// TwinCAT 3 PLC project Queque
// ProgramVersion: 3.1.0.9
// libraries:
//   CAA Memory, * (CAA Technical Workgroup)
//   VisuElem3DPath, 3.5.6.0 (System)
//   VisuElemMeter, 3.5.6.0 (System)
//   VisuElems, 3.5.6.10 (System)
//   VisuElemsDateTime, 3.5.6.0 (System)
//   VisuElemsSpecialControls, 3.5.6.0 (System)
//   VisuElemsWinControls, 3.5.6.0 (System)
//   VisuElemTextEditor, 3.5.6.0 (System)
//   visuinputs, 3.5.6.0 (system)
//   VisuNativeControl, 3.5.6.0 (System)
//   Tc2_MC2, * (Beckhoff Automation GmbH)
//   Tc2_Standard, * (Beckhoff Automation GmbH)
//   Tc2_System, * (Beckhoff Automation GmbH)
//   Tc2_TcpIp, * (Beckhoff Automation GmbH)
//   Tc2_Utilities, * (Beckhoff Automation GmbH)
//   Tc3_Interfaces, * (Beckhoff Automation GmbH)
//   Tc3_Module, * (Beckhoff Automation GmbH)
// project tree:
//   DUTs/enum/ ENUM_REC_FUNCTION_CODE.TcDUT
//   DUTs/struct/ ERROR_RECORD.TcDUT
//   / GlobalTextList.TcGTLO (not stored), PlcTask.TcTTO, Visualization Manager.TcVMO (not stored)
//   GVLs/ Error_Record_Data.TcGVL (not stored), MachineData.TcGVL (not stored)
//   POUs/AxisContrl/ Axis_Contrl.TcPOU
//   POUs/ CMD_Manage.TcPOU, Err_Record.TcPOU, IOInstances_Axis.TcPOU, IOInstances_Cylinder.TcPOU, MAIN.TcPOU (not stored), Param_Queue.TcGVL, P_TextModeWrite.TcPOU (not stored), Queue_REC_Contrl.TcPOU, Queue_SEND_Contrl.TcPOU
//   POUs/CMD_Manager_Ctrl/ CMD_Manager.TcPOU
//   POUs/CylinderContrl/ Cylinder_Contrl.TcPOU (not stored)
//   POUs/DUTs_Queue/ REC_CMD_DATA.TcDUT (not stored), REC_iCMD_DATA.TcDUT (not stored), SEND_CMD_DATA.TcDUT (not stored), SEND_iCMD_DATA.TcDUT
//   POUs/Queue_Ctrl/ Rec_Queue.TcPOU (not stored), Send_Queue.TcPOU (not stored)
//   POUs/TCP/ Client.TcPOU (not stored), Server.TcPOU
//   VISUs/ Axis_HMI_Struct.TcDUT, Axis_Page.TcVIS (not stored), CtrlMode_List.TcTLO, Cylinder.TcVIS, Cylinder_HMI_Structure.TcDUT (not stored), Err_record.TcVIS (not stored), Main.TcVIS

CONFIGURATION Queque
    RESOURCE PLC ON TwinCAT3
        TASK PlcTask(INTERVAL := T#10ms, PRIORITY := 20);
        PROGRAM MAIN WITH PlcTask : MAIN;
    END_RESOURCE
END_CONFIGURATION

// ---- DUTs/enum/ENUM_REC_FUNCTION_CODE.TcDUT
TYPE ENUM_REC_FUNCTION_CODE :
(
	(*__________Axis Control_________________*)
	MD  := 0,//Digital
	MA  := 1,//Analog
	G00 := 2,//move absolute
	G01 := 3,//move relative
	G02 := 4,//move velocity
	G03 := 5,//move Jog
	G04 := 6,//go home
	G05 := 7,//reset error
	G06 := 8,//stop
	
   (*________Cylinder Control_______________*)	
	C00 := 10,// Extend
	C01 := 11,// Retract
	C02 := 12 // Reset
)UDINT;
END_TYPE

// ---- DUTs/struct/ERROR_RECORD.TcDUT
TYPE ERROR_RECORD :
STRUCT
	Timer       : STRING;
	Axis        : UDINT;
	ErrorID     : UDINT;
	ErrorTXT    : STRING;
	ErrorCNT    : UDINT:=0;
END_STRUCT
END_TYPE

// ---- POUs/DUTs_Queue/SEND_iCMD_DATA.TcDUT
TYPE SEND_iCMD_DATA :
STRUCT
	DEVICE_ID       : UDINT;
	FUNCTIONCODE    : UDINT;
	DATA            : LREAL;
	Vel             : LREAL;
END_STRUCT
END_TYPE

// ---- VISUs/Axis_HMI_Struct.TcDUT
TYPE Axis_HMI_Struct :
STRUCT
	(*-------- input----------------*)
	mode                     : UDINT;
	bStop_Man                : BOOL;
	bHalt_Man                : BOOL;
	bReset_Man               : BOOL;
	bJog_F                   : BOOL;
	bJog_B                   : BOOL;
	bAbsGo_Man               : BOOL;
	bAddGo_Man               : BOOL;
	bVelGo_Man               : BOOL;
	bRelGo_Man               : BOOL;
	bModGo_Man               : BOOL;
	fSetAbsPos_Man           : LREAL;
	fSetRelPos_Man           : LREAL;
	fSetModPos_Man           : LREAL;
	fSetVel_Man              : LREAL;
	softLimitPOS_FW          : LREAL;
	softLimitPOS_BW          : LREAL;
	bForwordEnable           : BOOL;
	bBackwordEnable          : BOOL;
	bFW_LimitSwith           : BOOL;
	bBW_LimitSwith           : BOOL;
	bDog_PointSwith          : BOOL;

	(*---------output-------------*)
	bPowerEn                 : BOOL;
	bBusy                    : BOOL;
	bDone                    : BOOL;
	bAborted                 : BOOL;
	bError                   : BOOL;
	nErrorID                 : UDINT;
	cErrorTXT                : STRING;
	
	Axis_ref                 : Axis_ref;
END_STRUCT
END_TYPE

// ---- POUs/Param_Queue.TcGVL
VAR_GLOBAL CONSTANT
	MAX_QUEUE_SIZE : INT:= 10;

END_VAR

// ---- POUs/AxisContrl/Axis_Contrl.TcPOU
FUNCTION_BLOCK Axis_Contrl
VAR_IN_OUT
	HMI                      : Axis_HMI_Struct;
	Axis_CMD_Itf             : REC_CMD_DATA;
	Axis_ref                 : axis_ref;
END_VAR
VAR_INPUT
	mode                     : UDINT;
	bStop_Man                : BOOL;
	bStop_Auto               : BOOL;
	bHalt_Man                : BOOL;
	bReset_Man               : BOOL;
	bReset_Auto              : BOOL;
	bJog_F                   : BOOL;
	bJog_B                   : BOOL;
	bAbsGo_Man               : BOOL;
	bAbsGo_Auto              : BOOL;
	bVelGo_Man               : BOOL;
	bVelGo_Auto              : BOOL;
	bRelGo_Man               : BOOL;
	bRelGo_Auto              : BOOL;
	bModGo_Man               : BOOL;
	bModGo_Auto              : BOOL;
	bAddGo_Man               : BOOL;
	fSetAbsPos_Man           : LREAL;
	fSetAbsPos_Auto          : LREAL;
	fSetRelPos_Man           : LREAL;
	fSetRelPos_Auto          : LREAL;
	fSetModPos_Man           : LREAL;
	fSetModPos_Auto          : LREAL;
	fSetVel_Man              : LREAL;
	fSetVel_Auto             : LREAL;
	softLimitPOS_FW          : LREAL;
	softLimitPOS_BW          : LREAL;
	bForwordEnable           : BOOL:= TRUE;
	bBackwordEnable          : BOOL:= TRUE;
	bFW_LimitSwith           : BOOL:= TRUE;
	bBW_LimitSwith           : BOOL:= TRUE;
	bDog_PointSwith          : BOOL;
END_VAR
VAR_OUTPUT
	bPowerEn                 : BOOL;
	bBusy                    : BOOL;
	bDone                    : BOOL;
	bAborted                 : BOOL;
	bError                   : BOOL;
	nErrorID                 : UDINT;
	cErrorTXT                : STRING;
	nStatus                  : STRING;
END_VAR	
VAR

	mc_Stop                  : MC_Stop;
	mc_Reset                 : MC_Reset;
	mc_Power                 : MC_Power;
	mc_Jog                   : MC_Jog;
	mc_Home                  : MC_Home;
	mc_AbsMove               : MC_MoveAbsolute;
	mc_VelMove               : MC_MoveVelocity;
	mc_RelMove               : MC_MoveRelative;
	mc_ModMove               : MC_MoveModulo;
	mc_ReadAxisError         : MC_ReadAxisError;
	
	mc_AddMove               : MC_MoveAdditive;
	mc_Halt                  : MC_Halt;
	
	
	AbsMove_Rtrig            : R_Trig;
	VelMove_Rtrig            : R_Trig;
	RelMove_Rtrig            : R_Trig;
	ModMove_Rtrig            : R_Trig;

	
	AbsMove_state            : INT;
	VelMove_state            : INT;
	RelMove_state            : INT;
	ModMove_state            : INT;
	
	
	CMD_state                : UDINT;
END_VAR

Axis_AbsMove();
Axis_AddMove();
Axis_Home();
Axis_Jog();
Axis_ModMove();
Axis_Power();
Axis_RelMove();
Axis_Reset();
Axis_Stop();
Axis_VelMove();
HMI_Mapping();
Read_AxisError();
Axis_Halt();
Queue_Rec_Cmd();
//---------------------------------------
IF bError THEN
	nStatus:='ERROR';
ELSIF bDone AND (NOT bBusy) THEN
	nStatus:='DONE';
ELSIF Main.sReceiveData.Delete_Queue.FUNCTIONCODE = G05 THEN
	nStatus:= 'RESET DONE';
ELSE
	nStatus:= '';
END_IF

METHOD Axis_AbsMove
VAR_INPUT
END_VAR
mc_AbsMove( Axis:= Axis_ref );

IF ((bReset_Man OR bReset_Auto) AND (bError OR NOT mc_AbsMove.Busy)) 
	OR bStop_Auto OR bStop_Man  THEN
	mc_AbsMove.Execute:= FALSE;
	AbsMove_state:= 0;
END_IF

CASE mode OF
	1:
		mc_AbsMove.Position := fSetAbsPos_Man;
		mc_AbsMove.Velocity := ABS(fSetVel_Man);	
	2:
		mc_AbsMove.Position := fSetAbsPos_Auto;
		mc_AbsMove.Velocity := ABS(fSetVel_Auto);	
END_CASE

AbsMove_Rtrig(CLK:= ((mode = 1) AND bAbsGo_Man) OR ((mode = 2) AND bAbsGo_Auto) );

CASE AbsMove_state OF
	0:	
    	mc_AbsMove.Execute:= FALSE;
		IF AbsMove_Rtrig.Q THEN
			IF (NOT bForwordEnable) OR (NOT bBackwordEnable) 
				OR (mc_AbsMove.Position > softLimitPOS_FW) 
				OR (mc_AbsMove.Position < softLimitPOS_BW) 
				OR (NOT bFW_LimitSwith) OR (NOT bBW_LimitSwith)
				OR bError
				THEN
				bError:= TRUE;
				bBusy:= FALSE;
				bDone:= FALSE;
				bAborted:= FALSE;
				IF (NOT bForwordEnable) OR (NOT bBackwordEnable) THEN
					nErrorID:= 1;
					cErrorTXT:= 'Error: Axis not enable';
				ELSIF (mc_AbsMove.Position > softLimitPOS_FW) OR
					  (mc_AbsMove.Position < softLimitPOS_BW) THEN
					nErrorID:= 2;
					cErrorTXT:= 'Error: Axis Absolute Movement out of Limits';
				ELSIF (NOT bFW_LimitSwith) OR (NOT bBW_LimitSwith) THEN
					nErrorID:= 3;
					cErrorTXT:= 'Error: Axis reach limit swith';
				END_IF
			ELSE
				bBusy:= TRUE;
				bDone:= FALSE;
				bAborted:= FALSE;
				bError:= FALSE;
				nErrorID:= 0;
				cErrorTXT:= '';	
				AbsMove_state:= 1;
			END_IF
		END_IF
	1:
		mc_AbsMove.Execute:= TRUE;
		IF mc_AbsMove.Error THEN
			mc_AbsMove.Execute:= FALSE;
			bError:= TRUE;
			bAborted:= FALSE;
			bBusy:= FALSE;
			bDone:= FALSE;
			nErrorID:= DWORD_TO_UDINT (mc_AbsMove.ErrorID);
			cErrorTXT:= 'Error: Axis absolute movement error';
			AbsMove_state:= 0;
		ELSIF (NOT bFW_LimitSwith) OR (NOT bBW_LimitSwith) THEN
			mc_AbsMove.Execute:= FALSE;
			bError:= TRUE;
			bAborted:= FALSE;
			bBusy:= FALSE;
			bDone:= FALSE;
			nErrorID:= 3;
			cErrorTXT:= 'Error: Axis reach limit swith';
			AbsMove_state:= 0;
		ELSIF mc_AbsMove.Done THEN
			mc_AbsMove.Execute:= FALSE;
			bDone:= TRUE;
			bAborted:= FALSE;
			bBusy:= FALSE;
			AbsMove_state:= 0;
		ELSIF mc_AbsMove.CommandAborted THEN
			mc_AbsMove.Execute:= FALSE;
			bAborted:= TRUE;
			bDone:= FALSE;
			bBusy:= FALSE;
			AbsMove_state:= 0;
		END_IF
END_CASE
END_METHOD

METHOD Axis_AddMove
VAR_INPUT
END_VAR
mc_AddMove(
	Axis:=Axis_ref , 
	Execute:=bAddGo_Man , 
	Distance:=fSetRelPos_Man , 
	Velocity:= ABS(fSetVel_Man) , 
	Acceleration:= , 
	Deceleration:= , 
	Jerk:= , 
	BufferMode:= , 
	Options:= , 
	Done=> , 
	Busy=> , 
	Active=> , 
	CommandAborted=> , 
	Error=> , 
	ErrorID=> );
END_METHOD

METHOD Axis_Halt
VAR_INPUT
END_VAR
mc_Halt(
	Axis:= Axis_ref , 
	Execute:= bHalt_Man , 
	Deceleration:= , 
	Jerk:= , 
	BufferMode:= , 
	Options:= , 
	Done=> , 
	Busy=> , 
	Active=> , 
	CommandAborted=> , 
	Error=> , 
	ErrorID=> );
END_METHOD

METHOD Axis_Home
VAR_INPUT
END_VAR
mc_Home(
	Axis:= Axis_ref , 
	Position:= , 
	HomingMode:= MC_Direct , 
	bCalibrationCam:= bDog_PointSwith , 
	 );
	 
IF ((bReset_Man OR bReset_Auto) AND (bError OR NOT mc_Home.Busy)) 
	OR bStop_Auto OR bStop_Man  THEN
	mc_Home.Execute:= FALSE;
END_IF
END_METHOD

METHOD Axis_Jog
VAR_INPUT
END_VAR
mc_Jog(
	Axis:= Axis_ref , 
	JogForward:= bJog_F AND (mode = 1) AND bForwordEnable AND bFW_LimitSwith AND NOT bError , 
	JogBackwards:= bJog_B AND (mode = 1) AND bBackwordEnable AND bBW_LimitSwith AND NOT bError, 
	Mode:= MC_JOGMODE_CONTINOUS , 
	Position:= , 
	Velocity:= fSetVel_Man, 
	 );
END_METHOD

METHOD Axis_ModMove
VAR_INPUT
END_VAR
mc_ModMove( Axis:= Axis_ref , Direction:= MC_Shortest_Way );

IF ((bReset_Man OR bReset_Auto) AND (bError OR NOT mc_ModMove.Busy)) 
	OR bStop_Auto OR bStop_Man  THEN
	mc_ModMove.Execute:= FALSE;
	ModMove_state:= 0;
END_IF

CASE mode OF
	1:
		mc_ModMove.Velocity:= ABS(fSetVel_Man);
		mc_ModMove.Position:= fSetModPos_Man;
	2:
		mc_ModMove.Velocity:= ABS(fSetVel_Auto);
		mc_ModMove.Position:= fSetModPos_Auto;
END_CASE

ModMove_Rtrig(CLK:= ((mode = 1) AND bModGo_Man) OR ((mode = 2) AND bModGo_Auto) );

CASE ModMove_state OF
	0:
		mc_ModMove.Execute:= FALSE;
		IF ModMove_Rtrig.Q THEN
			IF (NOT bForwordEnable) OR (NOT bBackwordEnable) 
				OR (NOT bFW_LimitSwith) OR (NOT bBW_LimitSwith)
				OR bError
				THEN
				bError:= TRUE;
				bBusy:= FALSE;
				bDone:= FALSE;
				bAborted:= FALSE;
				IF (NOT bForwordEnable) OR (NOT bBackwordEnable) THEN
					nErrorID:= 1;
					cErrorTXT:= 'Error: Axis not enable';
				ELSIF (NOT bFW_LimitSwith) OR (NOT bBW_LimitSwith) THEN
					nErrorID:= 3;
					cErrorTXT:= 'Error: Axis reach limit swith';
				END_IF
			ELSE 
				bBusy:= TRUE;
				bDone:= FALSE;
				bAborted:= FALSE;
				bError:= FALSE;
				nErrorID:= 0;
				cErrorTXT:= '';	
				ModMove_state:= 1;
			END_IF
		END_IF
	1:
		mc_ModMove.Execute:= TRUE;
		IF mc_ModMove.Error THEN
			mc_ModMove.Execute:= FALSE;
			bError:= TRUE;
			bBusy:= FALSE;
			bDone:= FALSE;
			bAborted:= FALSE;
			nErrorID:= DWORD_TO_UDINT(mc_ModMove.ErrorID);
			cErrorTXT:= 'Error: Axis Modulo Movement error';
			ModMove_state:= 0;
		ELSIF (NOT bFW_LimitSwith) OR (NOT bBW_LimitSwith) THEN
			mc_AbsMove.Execute:= FALSE;
			bError:= TRUE;
			bAborted:= FALSE;
			bBusy:= FALSE;
			bDone:= FALSE;
			nErrorID:= 3;
			cErrorTXT:= 'Error: Axis reach limit swith';		
		ELSIF mc_ModMove.Done THEN
			mc_ModMove.Execute:= FALSE;
			bDone:= TRUE;
			bBusy:= FALSE;
			bAborted:= FALSE;
			ModMove_state:= 0;
		ELSIF mc_ModMove.CommandAborted THEN
			mc_ModMove.Execute:= FALSE;
			bAborted:= TRUE;
			bBusy:= FALSE;
			bDone:= FALSE;
			ModMove_state:= 0;
		END_IF
END_CASE
END_METHOD

METHOD Axis_Power
VAR_INPUT
END_VAR

mc_Power(
	Axis:= Axis_ref , 
	Enable:= TRUE , 
	Enable_Positive:= bFW_LimitSwith AND bForwordEnable , 
	Enable_Negative:= bBW_LimitSwith AND bBackwordEnable, 
	Override:=100.0 , 
	BufferMode:= , 
	Options:= , 
	Status=> bPowerEn , 
	Busy=> , 
	Active=> , 
	Error=> , 
	ErrorID=> );
END_METHOD

METHOD Axis_RelMove
VAR_INPUT
END_VAR
mc_RelMove(Axis:= Axis_ref);

IF ((bReset_Man OR bReset_Auto) AND (bError OR NOT mc_RelMove.Busy ))
	OR bStop_Man OR bStop_Auto THEN
	mc_RelMove.Execute:= FALSE;
	RelMove_state:= 0;
END_IF

CASE mode OF
	1:
		mc_RelMove.Velocity:= ABS(fSetVel_Man);
		mc_RelMove.Distance:= fSetRelPos_Man;
	2:
		mc_RelMove.Velocity:= ABS(fSetVel_Auto);
		mc_RelMove.Distance:= fSetRelPos_Auto;
END_CASE

RelMove_Rtrig(CLK:= ((mode = 1) AND bRelGo_Man) OR ((mode = 2) AND bRelGo_Auto) );

CASE RelMove_state OF
	0:
		mc_RelMove.Execute:= FALSE;
		IF RelMove_Rtrig.Q THEN
			IF (NOT bForwordEnable) OR (NOT bBackwordEnable) 
				OR ((mc_RelMove.Distance + Axis_ref.NcToPlc.ActPos) > softLimitPOS_FW) 
				OR ((mc_RelMove.Distance + Axis_ref.NcToPlc.ActPos) < softLimitPOS_BW)
				OR (NOT bFW_LimitSwith) OR (NOT bBW_LimitSwith)
				OR bError
				THEN
				bError:= TRUE;
				bAborted:= FALSE;
				bBusy:= FALSE;
				bDone:= FALSE;
				IF (NOT bForwordEnable) OR (NOT bBackwordEnable) THEN
					nErrorID:= 1;
					cErrorTXT:= 'Error: Axis not enable';
				ELSIF ((mc_RelMove.Distance + Axis_ref.NcToPlc.ActPos) > softLimitPOS_FW)
				    OR ((mc_RelMove.Distance + Axis_ref.NcToPlc.ActPos) < softLimitPOS_BW) THEN
					nErrorID:= 2;
					cErrorTXT:= 'Error: Axis Relative movement out of limits';
				ELSIF (NOT bFW_LimitSwith) OR (NOT bBW_LimitSwith) THEN
					nErrorID:= 3;
					cErrorTXT:= 'Error: Axis reach limit swith';
				END_IF
			ELSE
				bBusy:= TRUE;
				bDone:= FALSE;
				bAborted:= FALSE;
				bError:= FALSE;
				nErrorID:= 0;
				cErrorTXT:= '';	
				RelMove_state:= 1;
			END_IF
		END_IF
	1: 
		mc_RelMove.Execute:= TRUE;
		IF mc_RelMove.Error THEN
			mc_RelMove.Execute:= FALSE;
			bError:= TRUE;
			bAborted:= FALSE;
			bBusy:= FALSE;
			bDone:= FALSE;
			nErrorID:= DWORD_TO_UDINT(mc_RelMove.ErrorID);
			cErrorTXT:= 'Error: Axis Relative movement error';
			RelMove_state:= 0;
		ELSIF (NOT bFW_LimitSwith) OR (NOT bBW_LimitSwith) THEN
			mc_RelMove.Execute:= FALSE;
			bError:= TRUE;
			bAborted:= FALSE;
			bBusy:= FALSE;
			bDone:= FALSE;
			nErrorID:= 3;
			cErrorTXT:= 'Error: Axis reach limit swith';
		ELSIF mc_RelMove.Done THEN
			mc_RelMove.Execute:= FALSE;
			bDone:= TRUE;
			bAborted:= FALSE;
			bBusy:= FALSE;
			RelMove_state:= 0;
		ELSIF mc_RelMove.CommandAborted THEN
			mc_RelMove.Execute:= FALSE;
			bAborted:= TRUE;
			bBusy:= FALSE;
			bDone:= FALSE;
			RelMove_state:= 0; 
		END_IF 
		
END_CASE
END_METHOD

METHOD Axis_Reset
VAR_INPUT
END_VAR
mc_Reset( Axis:= Axis_ref);
IF bReset_Man OR bReset_Auto THEN
	IF mc_ReadAxisError.AxisErrorID <> 0 THEN	
		mc_Reset.Execute:= TRUE;
		IF mc_Reset.Done THEN
			mc_Reset.Execute:= FALSE;			
			bBusy:= FALSE;
			bDone:= FALSE;
			bAborted:= FALSE;
			bError:= FALSE;
			nErrorID:= 0;
			cErrorTXT:= '';
		END_IF
	ELSE
		mc_Reset.Execute:= FALSE;
			bBusy:= FALSE;
			bDone:= FALSE;
			bAborted:= FALSE;
			bError:= FALSE;
			nErrorID:= 0;
			cErrorTXT:= '';		
	END_IF
END_IF
END_METHOD

METHOD Axis_Stop
VAR_INPUT
END_VAR
mc_Stop( Axis:= Axis_ref );

IF bStop_Man OR bStop_Auto THEN
	mc_Stop.Execute:= TRUE;
	bStop_Man      := FALSE;
	bStop_Auto     := FALSE;
	bBusy          := FALSE;
	bAborted       := FALSE;
ELSE	
	mc_Stop.Execute:= FALSE;
END_IF

IF mc_Stop.Done THEN
	bDone  := TRUE;
END_IF
END_METHOD

METHOD Axis_VelMove
VAR
	fSetVelocity : LREAL;
END_VAR
mc_VelMove(Axis:= Axis_ref);

IF ((bReset_Man OR bReset_Auto) AND (bError OR NOT mc_VelMove.Busy)) 
	OR bStop_Auto OR bStop_Man  THEN	
	mc_VelMove.Execute:= FALSE;
	VelMove_state:= 0;
END_IF

CASE mode OF
	1:
		fSetVelocity:= fSetVel_Man;
	2:
		fSetVelocity:= fSetVel_Auto;
END_CASE

IF fSetVelocity >=0 THEN
	mc_VelMove.Direction:= MC_Positive_Direction;
ELSE
	mc_VelMove.Direction:= MC_Negative_Direction;	
END_IF

mc_VelMove.Velocity:= ABS(fSetVelocity);

VelMove_Rtrig(CLK:= ((mode = 1) AND bVelGo_Man ) OR ((mode = 2) AND bVelGo_Auto ));
CASE VelMove_state OF
	0:
		mc_VelMove.Execute:= FALSE;
		IF VelMove_Rtrig.Q THEN
			IF (NOT bForwordEnable) OR (NOT bBackwordEnable) 
				OR (NOT bFW_LimitSwith) OR (NOT bBW_LimitSwith)
				OR bError 
				THEN
				bError:= TRUE;
				bBusy:= FALSE;
				bDone:= FALSE;
				bAborted:= FALSE;
				IF (NOT bForwordEnable) OR (NOT bBackwordEnable) THEN
					nErrorID:= 1;
					cErrorTXT:= 'Error: Axis not enable';
				ELSIF (NOT bFW_LimitSwith) OR (NOT bBW_LimitSwith) THEN
					nErrorID:= 3;
					cErrorTXT:= 'Error: Axis reach limit swith';
				END_IF
			ELSE 
				bBusy:= TRUE;
				bDone:= FALSE;
				bAborted:= FALSE;
				bError:= FALSE;
				nErrorID:= 0;
				cErrorTXT:= '';	
				VelMove_state:= 1;
			END_IF
		END_IF
	1:
		mc_VelMove.Execute:= TRUE;
		IF mc_VelMove.Error THEN
			mc_VelMove.Execute:= FALSE;
			bError:= TRUE;
			bBusy:= FALSE;
			bDone:= FALSE;
			bAborted:= FALSE;
			nErrorID:= DWORD_TO_UDINT(mc_VelMove.ErrorID);
			cErrorTXT:= 'Error: Axis Velocity Movement error';
			VelMove_state:= 0;
		ELSIF mc_VelMove.InVelocity THEN//mc_Stop.Busy THEN
			mc_VelMove.Execute:= FALSE;
			bDone:= TRUE;
			bAborted:= FALSE;
			bBusy:= FALSE;			
			VelMove_state:= 0;
		ELSIF mc_VelMove.CommandAborted THEN
			mc_VelMove.Execute:= FALSE;
			bAborted:= TRUE;
			bBusy:= FALSE;
			bDone:= FALSE;
			VelMove_state:= 0; 
		END_IF
END_CASE
END_METHOD

METHOD HMI_Mapping
VAR_INPUT
END_VAR
(*---------------Input-------------------*)
mode                     := HMISwithMode;     
bStop_Man                := HMI.bStop_Man;  
bHalt_Man                := HMI.bHalt_Man;
bReset_Man               := HMI.bReset_Man;  
bJog_F                   := HMI.bJog_F;  
bJog_B                   := HMI.bJog_B;   
bAddGo_Man               := HMI.bAddGo_Man;
bAbsGo_Man               := HMI.bAbsGo_Man;  
bVelGo_Man               := HMI.bVelGo_Man;  
bRelGo_Man               := HMI.bRelGo_Man;  
bModGo_Man               := HMI.bModGo_Man; 
fSetAbsPos_Man           := HMI.fSetAbsPos_Man;
fSetRelPos_Man           := HMI.fSetRelPos_Man;
fSetModPos_Man           := HMI.fSetModPos_Man; 
fSetVel_Man              := HMI.fSetVel_Man; 
softLimitPOS_FW          := HMI.softLimitPOS_FW :=9999999999; 
softLimitPOS_BW          := HMI.softLimitPOS_BW :=-9999999999; 

(*---------------Output-------------------*)

HMI.bPowerEn              := bPowerEn;
HMI.bBusy                 := bBusy;
HMI.bDone                 := bDone;
HMI.bAborted              := bAborted;
HMI.bError                := bError;
HMI.nErrorID              := nErrorID;
HMI.cErrorTXT             := cErrorTXT;

HMI.bForwordEnable        := bForwordEnable; 
HMI.bBackwordEnable       := bBackwordEnable;  
HMI.bFW_LimitSwith        := bFW_LimitSwith;     
HMI.bBW_LimitSwith        := bBW_LimitSwith;
HMI.bDog_PointSwith       := bDog_PointSwith;

HMI.Axis_ref              := Axis_ref;
END_METHOD

METHOD Queue_Rec_Cmd
VAR_INPUT
END_VAR

CASE CMD_state OF
0:
	bAbsGo_Auto:=FALSE;
	bRelGo_Auto:=FALSE;
	bVelGo_Auto:=FALSE;
	bReset_Auto:=FALSE;
	bStop_Auto:=FALSE;
	CMD_state:=1;
1:
	IF Queue_RecDel_Flag THEN	
		CMD_state:=10;
		RETURN;
	END_IF

10:	
	CASE Axis_CMD_Itf.FUNCTIONCODE OF
		G00: //ABS
			bAbsGo_Auto:=TRUE;
			fSetAbsPos_Auto:=Axis_CMD_Itf.DATA;
			fSetVel_Auto:=Axis_CMD_Itf.Vel;
			CMD_state:=20;
		G01: //REL
			bRelGo_Auto:=TRUE;
			fSetRelPos_Auto:=Axis_CMD_Itf.DATA;
			fSetVel_Auto:=Axis_CMD_Itf.Vel;
			CMD_state:=20;
		G02: //VEL
			bVelGo_Auto:=TRUE;
			fSetVel_Auto:=Axis_CMD_Itf.Vel;
			IF mc_VelMove.InVelocity THEN
				CMD_state:=20;
			END_IF
		G03:
			CMD_state:=100;
		G04:
			CMD_state:=100;
		G05:// RESET
			CMD_state:=21;
			
		G06:// STOP
			bStop_Auto:=TRUE;	
			CMD_state:=20;
	ELSE
			CMD_state:=0;
	END_CASE
	
20:
	IF NOT bBusy THEN
		CMD_state:=100;		
	ELSIF bError THEN
		CMD_state:=0;
	END_IF
21:
	IF bError THEN
	bReset_Auto:=TRUE;
	CMD_state:=100;	
	END_IF
	IF NOT bError THEN
		CMD_state:=0;
	END_IF
	
100:	
	bAbsGo_Auto:=FALSE;
	bRelGo_Auto:=FALSE;
	bVelGo_Auto:=FALSE;
	bReset_Auto:=FALSE;
	bStop_Auto:=FALSE;
	CMD_state:=0;
END_CASE
END_METHOD

METHOD Read_AxisError
VAR_INPUT
END_VAR
mc_ReadAxisError(
	Axis:= Axis_ref, 
	Enable:= TRUE, 
	 );
IF mc_ReadAxisError.AxisErrorID <> 0 THEN
	bError:= TRUE;
	nErrorID:= DWORD_TO_UDINT(mc_ReadAxisError.AxisErrorID);
	cErrorTXT:= 'Error: Axis Drive Fault';
END_IF
END_METHOD

END_FUNCTION_BLOCK

// ---- POUs/CMD_Manage.TcPOU
FUNCTION_BLOCK CMD_Manage
VAR_INPUT

END_VAR
VAR_OUTPUT
END_VAR
VAR	
	CMD_state        : UDINT;
	SendDataDelay    : TON;
END_VAR

(*CASE CMD_state OF
0:
	Main.Axis.bAbsGo_Auto:=FALSE;
	Main.Axis.bRelGo_Auto:=FALSE;
	Main.Axis.bVelGo_Auto:=FALSE;
	Main.Axis.bReset_Auto:=FALSE;
	Main.Axis.bStop_Auto:=FALSE;
	
	Main.Cylinder.bExtend_auto:=FALSE;
	Main.Cylinder.bRetract_auto:=FALSE;
	Main.Cylinder.bReset_Error:= FALSE;
	
	Main.sSendData.bInsert:=FALSE;
	CMD_state:=1;
1:
	IF NOT Main.sReceiveData.Queue_Err THEN
		IF NOT  Main.sReceiveData.Queue_Empty THEN
			Main.sReceiveData.bDelete:= TRUE;
			CMD_state:=10;
		END_IF
	END_IF
	
10:	
	Main.sReceiveData.bDelete:= FALSE;
	CASE Main.sReceiveData.Delete_Queue.FUNCTIONCODE OF
		G00: //ABS
			Main.Axis.bAbsGo_Auto:=TRUE;
			Main.Axis.fSetAbsPos_Auto:=Main.sReceiveData.Delete_Queue.DATA;
			Main.Axis.fSetVel_Auto:=Main.sReceiveData.Delete_Queue.Vel;
			
			Main.sSendData.Insert_Queue.FUNCTIONCODE:=0;
			CMD_state:=20;
		G01: //REL
			Main.Axis.bRelGo_Auto:=TRUE;
			Main.Axis.fSetRelPos_Auto:=Main.sReceiveData.Delete_Queue.DATA;
			Main.Axis.fSetVel_Auto:=Main.sReceiveData.Delete_Queue.Vel;
			
			Main.sSendData.Insert_Queue.FUNCTIONCODE:=1;
			CMD_state:=20;
		G02: //VEL
			Main.Axis.bVelGo_Auto:=TRUE;
			Main.Axis.fSetVel_Auto:=Main.sReceiveData.Delete_Queue.Vel;
			
			Main.sSendData.Insert_Queue.FUNCTIONCODE:=2;
			CMD_state:=20;
		G03:
			Main.sSendData.Insert_Queue.FUNCTIONCODE:=3;
			CMD_state:=100;
		G04:
			Main.sSendData.Insert_Queue.FUNCTIONCODE:=4;
			CMD_state:=100;
		G05:// RESET
			Main.sSendData.Insert_Queue.FUNCTIONCODE:=5;
			CMD_state:=21;
			
		G06:// STOP
			Main.Axis.bStop_Auto:=TRUE;	
			
			Main.sSendData.Insert_Queue.FUNCTIONCODE:=6;
			CMD_state:=20;
			
		C00://Extend
			Main.Cylinder.bExtend_auto:= TRUE;
			
			Main.sSendData.Insert_Queue.FUNCTIONCODE:=7;
			Cmd_state:= 40;
		C01://Retract
			Main.Cylinder.bRetract_auto:= TRUE;
			
			Main.sSendData.Insert_Queue.FUNCTIONCODE:=8;
			Cmd_state:= 40;
		C02://reset
			Main.sSendData.Insert_Queue.FUNCTIONCODE:=9;
			Cmd_state:=41;
	ELSE
			CMD_state:=0;
	END_CASE
(*-------------------Axis----------------------------------*)	
20:
	Main.sSendData.Insert_Queue.STATUE:=Main.Axis.nStatus;
	IF Main.Axis.mc_VelMove.InVelocity THEN
		Main.sSendData.Insert_Queue.STATUE:='TRUE';
	END_IF
	IF NOT Main.sSendData.Queue_Err THEN
		IF NOT Main.sSendData.Queue_Full THEN
			Main.sSendData.bInsert:=TRUE;
		END_IF	
	END_IF
	CMD_state:=30;
	
21:
	IF Main.Axis.bError THEN
	Main.Axis.bReset_Auto:=TRUE;
	CMD_state:=31;
	ELSE
	CMD_state:= 0;
	END_IF	
	
30:
	IF NOT Main.Axis.bBusy THEN
		CMD_state:=100;				
	ELSIF Main.Axis.bError THEN
		CMD_state:=0;
	END_IF
	
31:
	IF NOT Main.Axis.bError THEN		
		Main.sSendData.Insert_Queue.STATUE:='TRUE';
	ELSE
		Main.sSendData.Insert_Queue.STATUE:=Main.Axis.nStatus;	
	END_IF
	IF NOT Main.sSendData.Queue_Err THEN
		IF NOT Main.sSendData.Queue_Full THEN
			Main.sSendData.bInsert:=TRUE;
		END_IF	
	END_IF
	CMD_state:=100;
	
(*----------------------------Cylinder-----------*)	
40:	
	Main.sSendData.Insert_Queue.STATUE:=Main.Cylinder.nStatus;
	IF NOT Main.sSendData.Queue_Err THEN
		IF NOT Main.sSendData.Queue_Full THEN
			Main.sSendData.bInsert:=TRUE;
		END_IF	
	END_IF
	Cmd_state:=50;
	
41:
	IF Main.Cylinder.error THEN
	Main.Cylinder.bReset_Error:= TRUE;
	Cmd_state:=51;
	END_IF	
50:
	IF Main.Cylinder.done THEN
		Cmd_state:=100;
	ELSE
		Cmd_state:=0;
	END_IF
	
51:
	IF NOT Main.Cylinder.error THEN
		Main.sSendData.Insert_Queue.STATUE:='TRUE';
	ELSE
		Main.sSendData.Insert_Queue.STATUE:=Main.Cylinder.nStatus;
	END_IF	
	IF NOT Main.sSendData.Queue_Err THEN
		IF NOT Main.sSendData.Queue_Full THEN
			Main.sSendData.bInsert:=TRUE;
		END_IF	
	END_IF
	Cmd_state:=100;
	
100:	
	Main.Axis.bAbsGo_Auto:=FALSE;
	Main.Axis.bRelGo_Auto:=FALSE;
	Main.Axis.bVelGo_Auto:=FALSE;
	Main.Axis.bReset_Auto:=FALSE;
	Main.Axis.bStop_Auto:=FALSE;
	Main.Cylinder.bExtend_auto:=FALSE;
	Main.Cylinder.bRetract_auto:=FALSE;
	Main.Cylinder.bReset_Error:= FALSE;
	
	Main.sSendData.bInsert:=FALSE;
	CMD_state:=0;
END_CASE

(*_______________Queue_send___________________*)
SendDataDelay(IN:=NOT SendDataDelay.Q , PT:=T#200MS , Q=> , ET=> );
IF SendDataDelay.Q THEN
	IF NOT Main.sSendData.Queue_Err THEN
		IF NOT Main.sSendData.Queue_Empty THEN
			Main.sSendData.bDelete:=TRUE;
		END_IF
	END_IF
ELSE
	Main.sSendData.bDelete:=FALSE;
END_IF *)

END_FUNCTION_BLOCK

// ---- POUs/CMD_Manager_Ctrl/CMD_Manager.TcPOU
FUNCTION_BLOCK CMD_Manager
VAR
	CMD_State     : UDINT;
	i             : UDINT;
	SendDataDelay : TON;
	StatueDelay   : TON;
	
END_VAR

CASE CMD_State OF
	0:
		Main.sSendData.bInsert:=FALSE;
		Main.sReceiveData.bDelete:= FALSE;
		Queue_RecDel_Flag:= FALSE;
		CMD_state:= 1;
	1:
		IF NOT Main.sReceiveData.Queue_Err THEN
			IF NOT  Main.sReceiveData.Queue_Empty THEN
				Main.sReceiveData.bDelete:= TRUE;
				Queue_RecDel_Flag:= TRUE;
				CMD_state:=10;
			//ELSE
				//CMD_state:=30; // wait statue
			END_IF
		END_IF
		
	10:
		Queue_RecDel_Flag:= FALSE;
		//ESTOP_BUTTON
		;
		//Machine Error
		;
		
		Main.sSendData.Insert_Queue.DEVICE_ID:= Main.sReceiveData.Delete_Queue.DEVICE_ID;
		Main.sSendData.Insert_Queue.FUNCTIONCODE := Main.sReceiveData.Delete_Queue.FUNCTIONCODE;
		Main.sSendData.Insert_Queue.STATUE :='';
		i := Main.sReceiveData.Delete_Queue.DEVICE_ID;	
		
		IF HMISwithMode = 1 THEN	
			Main.sSendData.Insert_Queue.STATUE :='Control Mode is Local Mode';
			CMD_State := 100;	
			RETURN;
		ELSE // Remote Mode,Find the difference instance device id
			IF (i >= 0) AND (i <=gDeviceCNT) THEN
				gDevice_ID[i]:=	Main.sReceiveData.Delete_Queue;
				Main.sSendData.Insert_Queue.STATUE :='CMD Have been received';
				IF NOT Main.sSendData.Queue_Err THEN
					IF NOT Main.sSendData.Queue_Full THEN
						Main.sSendData.bInsert:=TRUE;	
						CMD_State := 20;
						RETURN;
					END_IF	
				END_IF
			ELSE
				Main.sSendData.Insert_Queue.STATUE :='Error Device ID';
				CMD_State := 100;
				RETURN;
			END_IF
		END_IF
	20:
		Main.sSendData.bInsert:=FALSE;
		StatueDelay(IN:=TRUE , PT:=T#100MS , Q=> , ET=> );
		IF StatueDelay.Q THEN
			StatueDelay(IN:=FALSE );
			CMD_State := 30;
			RETURN;
		END_IF
	30:
	
		IF (gDevice_ID[i].Statue.STATUE = 'ERROR') OR (gDevice_ID[i].Statue.STATUE = 'DONE') OR (gDevice_ID[i].Statue.STATUE = 'RESET DONE')
		 THEN
		 	Main.sSendData.Insert_Queue.STATUE:= '';
			Main.sSendData.Insert_Queue.STATUE:=gDevice_ID[i].Statue.STATUE;
			CMD_State := 100;
			RETURN;
		//ELSE
			//Main.sSendData.Insert_Queue.STATUE :='Device ID Unuse now';
			//CMD_State := 0;
			//RETURN;
		END_IF
	
	100:// Insert data to SendQueue
		IF NOT Main.sSendData.Queue_Err THEN
			IF NOT Main.sSendData.Queue_Full THEN
				Main.sSendData.bInsert:=TRUE;	
				CMD_State := 0;
				RETURN;
			END_IF	
		END_IF
ELSE
	CMD_State := 0;		
END_CASE



(*_______________Queue_send___________________*)
	

IF NOT Main.sSendData.Queue_Err THEN
	IF NOT Main.sSendData.Queue_Empty THEN
		Main.sSendData.bDelete:=TRUE;	
	ELSE
		Main.sSendData.bDelete:=FALSE;
	END_IF
END_IF

END_FUNCTION_BLOCK

// ---- POUs/Err_Record.TcPOU
FUNCTION_BLOCK Err_Record

VAR
	fbGetLocalTime      : NT_GetTime;
	RecordTime          : STRING;
	Init_List           : ERROR_RECORD;
	RecordR_TRIG        : R_TRIG;
	j                   : UDINT:=0;
	AxisErrCNT          : UDINT:=0;
END_VAR

(*------------------------local time-------------------------*)
fbGetLocalTime();
IF fbGetLocalTime.START  THEN
	fbGetLocalTime.START:=FALSE;
	RecordTime:=SYSTEMTIME_TO_STRING(fbGetLocalTime.TIMESTR);
ELSE
	fbGetLocalTime.START:=TRUE;
END_IF

(*--------------------------Error count-----------------------*)
AxisErrCNT:=0;
FOR j:=gAxisBeginNum TO gAxisEndNum BY 1 DO	
	RecordR_TRIG(CLK:= gAxisCtrl[j].bError);	
END_FOR
IF RecordR_TRIG.Q THEN
	IF gAxisCtrl[j].bError THEN	
		i:=i+1;
		Error_List[i].Timer:=RecordTime;
		Error_List[i].Axis:= j;
		Error_List[i].ErrorID:= gAxisCtrl[j].nErrorID;
		Error_List[i].ErrorTXT:=gAxisCtrl[j].cErrorTXT;
		Error_List[i].ErrorCNT:=i; 	
	END_IF
END_IF	

(*(RecordR_TRIG(CLK:= gAxisCtrl[j].bError);
IF RecordR_TRIG.Q THEN
	IF gAxisCtrl[j].bError THEN	
		i:=i+1;
		Error_List[i].Timer:=RecordTime;
		Error_List[i].ErrorID:= gAxisCtrl[j].nErrorID;
		Error_List[i].ErrorTXT:=gAxisCtrl[j].cErrorTXT;
		Error_List[i].ErrorCNT:=i; 
	IF gCylinderCtrl[j].error THEN
		i:=i+1;
		Error_List[i].Timer:=RecordTime;
		Error_List[i].ErrorID:=gCylinderCtrl[j].errorID;
		Error_List[i].ErrorTXT:=gCylinderCtrl[j].errorTXT;	
		Error_List[i].ErrorCNT:=i;	 
	END_IF
END_IF  *)


IF i=MAX_ERROR_SIZE THEN
	FOR i:=1 TO MAX_ERROR_SIZE BY 1
	DO
		Error_List[i]:=Init_List;
	END_FOR
	i:=0;
END_IF

END_FUNCTION_BLOCK

// ---- POUs/IOInstances_Axis.TcPOU
PROGRAM IOInstances_Axis
VAR
END_VAR

gAxisCtrl[1](
	HMI:= gAxisCtrl_HMI[1] , 
	Axis_CMD_Itf:= gDevice_ID[1]  , 
	Axis_ref:= gAxis[1] ,
	mode:= , 
	bStop_Man:= , 
	bStop_Auto:= , 
	bHalt_Man:= , 
	bReset_Man:= , 
	bReset_Auto:= , 
	bJog_F:= , 
	bJog_B:= , 
	bAbsGo_Man:= , 
	bAbsGo_Auto:= , 
	bVelGo_Man:= , 
	bVelGo_Auto:= , 
	bRelGo_Man:= , 
	bRelGo_Auto:= , 
	bModGo_Man:= , 
	bModGo_Auto:= , 
	bAddGo_Man:= , 
	fSetAbsPos_Man:= , 
	fSetAbsPos_Auto:= , 
	fSetRelPos_Man:= , 
	fSetRelPos_Auto:= , 
	fSetModPos_Man:= , 
	fSetModPos_Auto:= , 
	fSetVel_Man:= , 
	fSetVel_Auto:= , 
	softLimitPOS_FW:= , 
	softLimitPOS_BW:= , 
	bForwordEnable:= , 
	bBackwordEnable:= , 
	bFW_LimitSwith:= , 
	bBW_LimitSwith:= , 
	bDog_PointSwith:= , 
	bPowerEn=> , 
	bBusy=> , 
	bDone=> , 
	bAborted=> , 
	bError=> , 
	nErrorID=> , 
	cErrorTXT=> , 
	nStatus=>gDevice_ID[1].Statue.STATUE );

END_PROGRAM

// ---- POUs/IOInstances_Cylinder.TcPOU
PROGRAM IOInstances_Cylinder
VAR
END_VAR

gCylinderCtrl[30](
	Cylinder_HMI:= gCylinderCtrl_HMI[30]  , 
	Cylinder_CMD_Itf:= gDevice_ID[30], 
	mode:= , 
	bExtend_auto:= , 
	bRetract_auto:= , 
	bExtend_jog:= , 
	bRetract_jog:= , 
	bExtend_Enable:= , 
	bRetract_Enable:= , 
	bAbort_Enable:= , 
	bExtend_Prox:= , 
	bRetract_Prox:= , 
	bReset_Error:= , 
	tTimeOut:= , 
	bExtend_Work=> , 
	bRetract_Work=> , 
	done=> , 
	busy=> , 
	error=> , 
	errorID=> , 
	errorTXT=> , 
	doneCNT=> , 
	errorCNT=> , 
	nStatus=>gDevice_ID[30].Statue.STATUE );

END_PROGRAM

// ---- POUs/Queue_REC_Contrl.TcPOU
FUNCTION_BLOCK Queue_REC_Contrl
VAR
	REC_Queue_List      : ARRAY[0..Param_Queue.MAX_QUEUE_SIZE] OF REC_CMD_DATA;
	REC_Queue           : Rec_Queue;
	
	Head_Queue          : REC_CMD_DATA;	
	
	InsertR_TRIG        : R_TRIG;
	DeleteR_TRIG        : R_TRIG;
	InitR_TRIG          : R_TRIG;
	

	
	bInit               : BOOL;
	
	Queue_CNT           : INT;
	Queue_Full          : BOOL;
	Queue_Empty         : BOOL;
	Queue_Err           : BOOL;
	
		
END_VAR
VAR_INPUT
	Insert_Queue        : REC_CMD_DATA;
	Delete_Queue        : REC_CMD_DATA;
	bInsert             : BOOL;
	bDelete             : BOOL;
END_VAR

REC_Queue(REC_Queue_List:=REC_Queue_List , Err_Out=>Queue_Err );

Head_Queue:= REC_Queue.Head_Queue();
Queue_CNT:= REC_Queue.Count_Queue();
Queue_Full:= REC_Queue.Full_Queue();
Queue_Empty:= REC_Queue.Empty_Queue();

InsertR_TRIG(CLK:= bInsert);
IF InsertR_TRIG.Q THEN
	REC_Queue.Insert_Queue(Insert_Queue:= Insert_Queue);
END_IF

DeleteR_TRIG(CLK:= bDelete);
IF DeleteR_TRIG.Q THEN
	Delete_Queue:= REC_Queue.Delete_Queue();
END_IF

InitR_TRIG(CLK:= bInit);
IF InitR_TRIG.Q THEN
	REC_Queue.Init_Queue();
END_IF

END_FUNCTION_BLOCK

// ---- POUs/Queue_SEND_Contrl.TcPOU
FUNCTION_BLOCK Queue_SEND_Contrl
VAR
	SEND_Queue_List     : ARRAY[0..Param_Queue.MAX_QUEUE_SIZE] OF SEND_CMD_DATA;
	SEND_Queue          : Send_Queue;	
	Head_Queue          : SEND_CMD_DATA;
	
	InsertR_TRIG        : R_TRIG;
	DeleteR_TRIG        : R_TRIG;
	InitR_TRIG          : R_TRIG;
	
	
	bInit               : BOOL;
	
	Queue_CNT           : INT;
	Queue_Full          : BOOL;
	Queue_Empty         : BOOL;
	Queue_Err           : BOOL;
END_VAR
VAR_INPUT
	Insert_Queue        : SEND_CMD_DATA;
	Delete_Queue        : SEND_CMD_DATA;
	bInsert             : BOOL;
	bDelete             : BOOL;
END_VAR

SEND_Queue(SEND_Queue_List:=SEND_Queue_List , Err_Out=>Queue_Err );

Head_Queue:= SEND_Queue.Head_Queue();
Queue_CNT:= SEND_Queue.Count_Queue();
Queue_Full:= SEND_Queue.Full_Queue();
Queue_Empty:= SEND_Queue.Empty_Queue();

InsertR_TRIG(CLK:= bInsert);
IF InsertR_TRIG.Q THEN
	SEND_Queue.Insert_Queue(Insert_Queue:= Insert_Queue);
END_IF

DeleteR_TRIG(CLK:= bDelete);
IF DeleteR_TRIG.Q THEN	
	Delete_Queue:= SEND_Queue.Delete_Queue();
	Queue_SendDel_Flag:= TRUE;
ELSE
	Queue_SendDel_Flag:= FALSE;
END_IF

InitR_TRIG(CLK:= bInit);
IF InitR_TRIG.Q THEN
	SEND_Queue.Init_Queue();
END_IF

END_FUNCTION_BLOCK

// ---- POUs/TCP/Server.TcPOU
FUNCTION_BLOCK Server
VAR_INPUT
	sLocalHost         : T_IPv4AddR;
	nLocalPort         : UDINT;         
    bConnectEnable     : BOOL;  
	bRestart_Connect   : BOOL;        
	bSendExecute       : BOOL;
	sSendData          : SEND_CMD_DATA;//STRING(255);
END_VAR
VAR_OUTPUT
	eState             : E_SocketConnectionState;
	bReceiveDone       : BOOL;
	sReceiveData       : REC_CMD_DATA;//STRING(255);
END_VAR
VAR
	bCreateServerHnd   : BOOL;
	bRestart_Connect_Flag : BOOL;
	FB_Connection      : FB_ServerClientConnection;
	FB_SocketSend      : FB_SocketSend;
	FB_SocketReceive   : FB_SocketReceive;
	FB_SocketClose     : FB_SocketClose;
	
	sSrvNetID          : T_AmsNetID:='';
	hServer            : T_HSERVER;
	hSocket            : T_HSOCKET;
	sRemoteHost        : T_IPv4Addr;
	nRemoteport        : UDINT;
	sSendDataTemp      : SEND_CMD_DATA;//STRING(255);	
	sSendDataInit      : SEND_CMD_DATA;
	sReceiveDataTemp   : REC_CMD_DATA;//STRING(255);
	sReceiveDataInit   : REC_CMD_DATA;
	
	nState             : INT;
	tSendDalay         : TON;
	tReceiveDalay      : TON;
	tRestartDalay      : TON;
	SendRtrig          : R_TRIG;
	RestartRtrig       : R_TRIG;
END_VAR

tRestartDalay(IN:= (bRestart_Connect AND hSocket.handle >0) , PT:= T#2S);
RestartRtrig(CLK:= tRestartDalay.Q );
IF RestartRtrig.Q THEN
	bRestart_Connect_Flag := TRUE;
END_IF

bCreateServerHnd:= F_CreateServerHnd(
										sSrvNetID:=sSrvNetID , 
										sLocalHost:=sLocalHost , 
										nLocalPort:=nLocalPort , 
										nMode:=LISTEN_MODE_CLOSEALL OR CONNECT_MODE_ENABLEDBG , 
										bEnable:=TRUE , 
										hServer:=hServer );

FB_Connection(
	hServer:=hServer , 
	eMode:=eACCEPT_ALL , 
	sRemoteHost:=sRemoteHost , 
	nRemotePort:=nRemoteport , 
	bEnable:=bConnectEnable AND bCreateServerHnd AND (NOT FB_SocketClose.bBusy) , 
	tReconnect:=T#1S , 
	bBusy=> , 
	bError=> , 
	nErrID=> , 
	hSocket=>hSocket , 
	eState=>eState );
	
FB_SocketSend(
	sSrvNetId:=sSrvNetID , 
	hSocket:=hSocket , 
	cbLen:=SIZEOF(sSendDataTemp), 
	pSrc:=ADR(sSendDataTemp) , 
	bExecute:= , 
	tTimeout:=T#5S , 
	bBusy=> , 
	bError=> , 
	nErrId=> );

FB_SocketReceive(
	sSrvNetId:=sSrvNetID , 
	hSocket:=hSocket , 
	cbLen:=SIZEOF(sReceiveDataTemp) , 
	pDest:=ADR(sReceiveDataTemp) , 
	bExecute:= , 
	tTimeout:=T#5S , 
	bBusy=> , 
	bError=> , 
	nErrId=> , 
	nRecBytes=> );
	
FB_SocketClose(
	sSrvNetId:=sSrvNetID , 
	hSocket:=hSocket , 
	bExecute:= , 
	tTimeout:=T#5S , 
	bBusy=> , 
	bError=> , 
	nErrId=> );
	
CASE nState OF
	0: 
		IF bRestart_Connect_Flag THEN
			bRestart_Connect_Flag:= FALSE;
			FB_SocketClose.bExecute:= FALSE;
			nState:= 10;
		ELSE
			bRestart_Connect_Flag:= FALSE;
			nState:=1;
		END_IF
	1:
		IF hSocket.handle > 0 AND (eState = eSocket_Connected) THEN
			tReceiveDalay(IN:=NOT tReceiveDalay.Q , PT:=T#10MS , Q=> , ET=> );	
			IF tReceiveDalay.Q THEN
				tReceiveDalay(IN:=FALSE);
				FB_SocketReceive.bExecute:=TRUE;
				nState:=2;
			END_IF
		END_IF
	2:
		FB_SocketReceive.bExecute:=FALSE;
		IF NOT FB_SocketReceive.bBusy THEN
			IF NOT FB_SocketReceive.bError THEN
				IF FB_SocketReceive.nRecBytes <> 0 THEN
					sReceiveData:=sReceiveDataInit;
					sReceiveData:=sReceiveDataTemp;//LEFT(cReceiveDataTemp,UDINT_TO_INT(FB_SocketReceive.nRecBytes));
					bReceiveDone:=TRUE;
					nState:=0;
				ELSE
					bReceiveDone:= FALSE;				
					sReceiveDataTemp:= sReceiveDataInit;
					nState:= 0;
				END_IF
			ELSE 
				FB_SocketClose.bExecute:=FALSE;
				nState :=10;
			END_IF
		END_IF
	10:
		FB_SocketClose.bExecute:=TRUE;
		nState :=20;
	20:
		IF FB_SocketClose.bBusy THEN
			IF FB_SocketClose.bError THEN
				nState:=0;
			ELSE
				nState:=10;
			END_IF
			FB_SocketClose.bExecute:=FALSE;
		END_IF
		
END_CASE

//tSendDalay(IN:=NOT tSendDalay.Q , PT:=T#200MS , Q=> , ET=> );
SendRtrig(CLK:=bSendExecute);
IF SendRtrig.Q AND (NOT FB_SocketSend.bBusy) THEN
	sSendDataTemp:=sSendDataInit;
	sSendDataTemp:=sSendData;
	FB_SocketSend.bExecute:=TRUE;
ELSE
	FB_SocketSend.bExecute:=FALSE;
END_IF

END_FUNCTION_BLOCK

// ---- VISUs/CtrlMode_List.TcTLO
TEXTLIST CtrlMode_List
  1 = 'Local Mode'
  2 = 'Remote Mode'
   = ''
END_TEXTLIST

// ---- VISUs/Cylinder.TcVIS
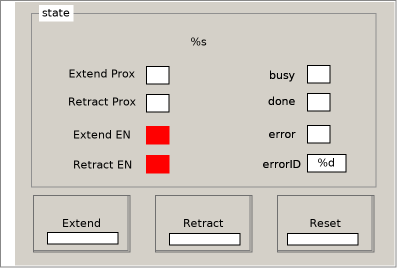
VISUALIZATION Cylinder  // 397x268
VAR_IN_OUT
	userdata : Cylinder_HMI_Structure;
END_VAR
    Rectangle (14,1 381x265)
    GroupBox (31,5 345x182), "state"
        Rectangle (276,60 23x18), colour toggle: userData.busy
        Rectangle (276,88 23x18), colour toggle: userData.done
        Rectangle (276,120 23x18), colour toggle: userData.error
        Rectangle (276,149 39x18), "%d", text variable: userData.errorID, colour toggle: userData.errorID
        Rectangle (115,61 23x18), colour toggle: userData.bExtend_Prox
        Rectangle (115,89 23x18), colour toggle: userData.bRetract_Prox
        Rectangle (115,121 23x18), colour toggle: userData.bExtend_Enable
        Label (191,52 120x37), "busy"
        Label (191,78 120x37), "done"
        Label (191,111 120x37), "error"
        Label (191,141 120x37), "errorID"
        Rectangle (115,150 22x18), colour toggle: userData.bRetract_Enable
    Rectangle (62,27 273x30), "%s", text variable: userData.errorTXT, colour toggle: userData.errorTXT
    Rectangle (307,65 23x18), colour toggle: userData.busy
    Rectangle (307,93 23x18), colour toggle: userData.done
    Rectangle (307,125 23x18), colour toggle: userData.error
    Rectangle (307,154 39x18), "%d", text variable: userData.errorID, colour toggle: userData.errorID
    Rectangle (146,66 23x18), colour toggle: userData.bExtend_Prox
    Rectangle (146,94 23x18), colour toggle: userData.bRetract_Prox
    Rectangle (146,126 23x18), colour toggle: userData.bExtend_Enable
    Label (222,57 120x37), "busy"
    Label (222,83 120x37), "done"
    Label (222,116 120x37), "error"
    Label (222,146 120x37), "errorID"
    Rectangle (146,155 23x18), colour toggle: userData.bRetract_Enable
    Group (33,195 97x57)
        Button (0,0 97x57), "Extend"
            tap userData.bExtend_jog
        Rectangle (14,37 71x12), colour toggle: userData.bExtend_Work
    Group (155,195 97x57)
        Button (0,0 97x57), "Retract"
            tap userData.bRetract_jog
        Rectangle (14,38 71x12), colour toggle: userData.bRetract_Work
    Group (277,195 97x57)
        Button (0,0 97x57), "Reset"
            tap userData.bReset_Error
        Rectangle (10,38 71x12), colour toggle: userData.error
    Group (27,59 150x121)
        Label (0,0 150x30), "Extend Prox"
        Label (0,28 150x30), "Retract Prox"
        Label (0,61 150x30), "Extend EN"
        Label (1,91 149x30), "Retract EN"
END_VISUALIZATION

// ---- VISUs/Main.TcVIS
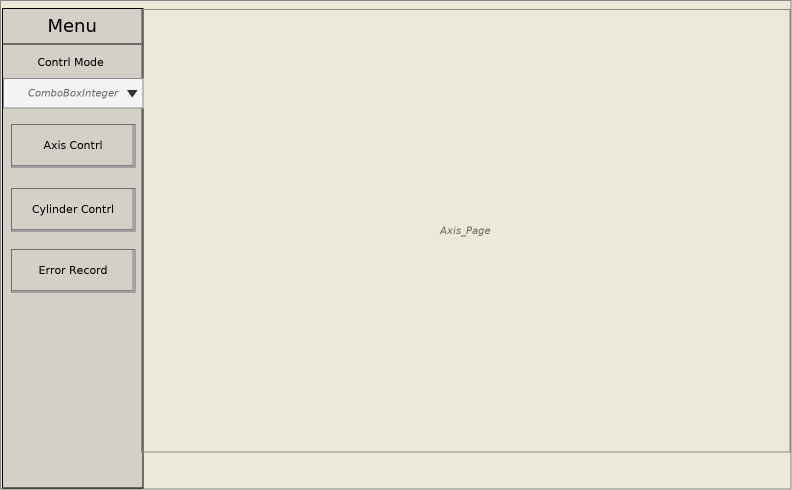
VISUALIZATION Main  // 792x490
    Rectangle (2,8 141x480)
    Rectangle (2,8 141x36), "Menu"
    Rectangle (4,46 134x33), "Contrl Mode"
    Button (11,124 124x43), "Axis Contrl"
        OnMouseDown: FrameSelectionChange Selection=SelectedFrame=54291640-e5ed-4e41-8a36-41169059765e, GlobSel=AssignType=Directly, SelType=Locally
    Button (11,188 124x43), "Cylinder Contrl"
        OnMouseDown: FrameSelectionChange Selection=SelectedFrame=54291640-e5ed-4e41-8a36-41169059765e, Selection=1, GlobSel=AssignType=Directly, SelType=Locally
    Frame (141,9 649x443)
        shows Axis_Page(userdata := gAxisCtrl_HMI[1])
        shows Cylinder(userdata := gCylinderCtrl_HMI[30])
        shows Err_record()
    ComboBoxInteger (3,78 140x30), variable: HMISwithMode, text list: 'CtrlMode_List'
    Button (11,249 124x43), "Error Record"
        OnMouseDown: FrameSelectionChange Selection=SelectedFrame=54291640-e5ed-4e41-8a36-41169059765e, Selection=2, GlobSel=AssignType=Directly, SelType=Locally
END_VISUALIZATION
